Fanuc KAREL source: ka00133.KL

-- PROVISIONAL review KL for V940-1; original PC SHA256 4ec96f16cceeba01c4a84bf18a2768b53e71f0cc3fce08f6c91491aaee9407a0
-- Incomplete behavior may be omitted. Consult companion uncertainty JSON. Do not deploy.
PROGRAM KA00133
%NOLOCKGROUP
VAR
  DST : INTEGER
-- UNRESOLVED_DECL SRC type=002017
BEGIN
  -- V9_ZERO_TABLE_METADATA_HINT layout=0001; no indexed target words; source/name/runtime held
  -- UNRESOLVED_PC offsets 5-19; opcodes 2E,22,9D,33,B4
  -- UNRESOLVED_PC offsets 24-39; opcodes 22,9D,33,B3,23
  -- UNRESOLVED_PC offsets 44-48; opcodes 7F
END KA00133
